// TwinCAT 3 PLC project TrainingPLC2
// ProgramVersion: 3.1.4024.0
// libraries:
//   Tc2_Standard, * (Beckhoff Automation GmbH)
//   Tc2_System, * (Beckhoff Automation GmbH)
//   Tc3_Module, * (Beckhoff Automation GmbH)
//   VisuSymbols,3.5.10.0,System
// project tree:
//   / GlobalTextList.TcGTLO, PlcTask.TcTTO, Visualization Manager.TcVMO (not stored)
//   POUs/ MAIN.TcPOU, NEWSUBROUTINE.TcPOU, notes.TcPOU, CalculateSine.TcPOU, prgPumpControl.TcPOU
//   VISUs/ Visualization.TcVIS
// real-time tasks:
//   TASK PlcTask: cycle T#10ms, priority 20, ADS port 350
//   TASK PlcTask1: cycle T#10ms, priority 21, ADS port 351

CONFIGURATION TrainingPLC2
    RESOURCE PLC ON TwinCAT3
        TASK PlcTask(INTERVAL := T#10ms, PRIORITY := 20);
        PROGRAM MAIN WITH PlcTask : MAIN;
    END_RESOURCE
END_CONFIGURATION

// ---- POUs/MAIN.TcPOU
PROGRAM MAIN
VAR
	counter : REAL := 1;
	toggle: BOOL;
	pushButton	:BOOL;
	clickButton :BOOL;
	light 		:BOOL;
	t1 			:TON;
	tr1			:R_TRIG;
	pulse		:TP;
	
	sine		:REAL;
END_VAR

prgPumpControl();
IF counter > 4000 THEN
	counter := 0;
ELSE
	counter := counter+1;
END_IF

sine := SIN(counter/500);




//counter:= counter+2;

//t1(IN:=pushButton, PT:= T#5S, Q=> light, ET=> );
//t1(PT:= T#5S );
//t1.IN:=pushButton;

//pulse(IN:= pushButton, PT:= T#500MS, Q=> , ET=> ); 
//tr1(CLK:= clickButton, Q=> light);

//IF counter > 1000 THEN
//	counter := 0;
//	toggle := NOT toggle;
	
//	NEWSUBROUTINE(input:=toggle);
//	//comment
//	(*
//	multi
//	line 
//	comment
//	*)
//END_IF

ACTION ACT:
// NETWORK 1
END_ACTION

END_PROGRAM

// ---- POUs/prgPumpControl.TcPOU
PROGRAM prgPumpControl
VAR
	bStart_PB	AT %I* :BOOL;
	bStop_PB	AT %I* :BOOL;
	bPumpRelay	AT %Q* :BOOL;
END_VAR

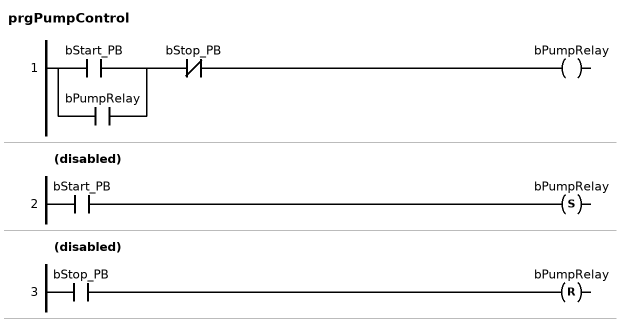
// NETWORK 1
bPumpRelay := (bStart_PB OR bPumpRelay) AND NOT bStop_PB;

// NETWORK 2 (disabled)
// bPumpRelay S= bStart_PB;

// NETWORK 3 (disabled)
// bPumpRelay R= bStop_PB;

END_PROGRAM

// ---- POUs/NEWSUBROUTINE.TcPOU
PROGRAM NEWSUBROUTINE

VAR_INPUT
	input	:BOOL;	
END_VAR
VAR
	c1		:CTD;
	counter2 :LREAL:=3.5;
	
END_VAR

//c1(
//	CD:= , 
//	LOAD:= , 
//	PV:= , 
//	Q=> , 
//	CV=> );


//IF input = TRUE THEN
//	counter2 := counter2 + 1;
//ELSE
//	counter2 := counter2 - 1;
//END_IF

END_PROGRAM

// ---- POUs/notes.TcPOU
PROGRAM notes
VAR
END_VAR

(*


https://docs.google.com/document/d/1TtsSPKcGf5wqr-mFV1IPG9VzqW2f_MM_MVhuRm0hRRs/edit?tab=t.0



To add a shortcut:
1. Tools -> Options -> Environment -> Keyboard
2. Search for functions
	Example: Logintonone
3. Press shortcut keys -> Assign



Change variables while running program
1. Add value to 'prepared values' column
2. 'Write values' (top right)
	Shortcut -> Alt-W 
	
	
Shortcuts:
Write values: Alt-W
Login: Alt-X
Logout: Alt-Z
Input assistant: F2 (or right click in program section

Terms:
Rising edge: when input goes from low to high
Falling edge: opposite of above

Notes:
Libraries are in PLC -> references
Set reserved/shared cores in SYSTEM-> Real-Time
Set run speed (cycles) in PLC -> PlcTask, or SYSTEM -> Tasks -> PlcTask
Multi line comments  -> (**)
Regular comment -> /

if statement:
IF {condition} THEN
	{body}
END_IF

loop:
FOR variable := start-value TO end-value [ BY step-value ] DO
    statement;
    statement;
    ..
    statement;
END_FOR;

function:
Function CalcStdDev : LREAL
var_input v1,v2,v3,v4 : LREAL; end_var

var 
    SumOfSquares : LREAL;
    Mean : LREAL;
end_var

    (* Calculate the mean *)
    Mean := (v1 + v2 + v3 + v4) / 4;

    (* Calculate the standard deviation *)
    SumOfSquares := (v1 - Mean) ** 2 +
                (v2 - Mean) ** 2 +
                (v3 - Mean) ** 2 +
                (v4 - Mean) ** 2;

    CalcStdDev := sqrt( SumOfSquares / 4 );
End_Function



INPUT VARIABLE
var AT %I* : TYPE
OUTPUT VARIABLE
var AT %Q* : TYPE


Variable types
BOOL
INTEGER
- BYTE
- WORD
- DWORD
- LWORD
more common
- SINT
- INT
- DINT
- LINT
- U+^ (unsigned)
FLOATING POINT
- REAL (32 bit)
- LREAL (64 bit)
TIME
- TIME (T#5d5h5m5s5ms)
- LTIME (LTIME#5d5h5m5s5ms5us5ns)
DATE
- LOTS (D#xxxx)
STRING
more
BIT
POINTER
REFERENCE
UNION
ANY
+user data types


all are 0 (or false) by default
constants 
VAR CONSTANT
	(must be assigned)
END_VAR


*)

END_PROGRAM

// ---- POUs/CalculateSine.TcPOU
FUNCTION CalculateSine : REAL
VAR_INPUT
	angle_in_radians : REAL;
END_VAR

VAR_OUTPUT
	sine_value : REAL;
END_VAR

sine_value := SIN(angle_in_radians);

END_FUNCTION

// ---- VISUs/Visualization.TcVIS
VISUALIZATION Visualization  // 2x2
END_VISUALIZATION
